Staubli VAL3: Motion.dtx

mdesc mNomSpeed
bool bPause
bool bRuning
bool bStop
tool tTool = {fatherId=flange[0], ioLink=valve1}
frame fFrame = {fatherId=world[0]}
pointRx pDemo = {fatherId=fFrame[0]}
string sFolder = "Disk://Traj/"
string sPtpara
configRx cConfig
num l_nRes
bool bExit
bool bUserRefresh
bool bListRefresh
string sPath
string sList
num nSelected
string sItem
string sProductList
pointRx pPoint = {fatherId=world[0]}
pointRx pSparePoint = {fatherId=world[0]}
string sMsg[8]
